// TIA Portal V19 export
FUNCTION "CallAck" : Void   // FC2, LAD
// stored: SetENOAutomatically false
BEGIN
END_FUNCTION
